TYPE ST_InternalPowerSupply_Params :
STRUCT
	i_ACStartupDelay : INT := 100; //ms
	i_DCPSU_StartupDelay: INT := 1000; //ms
	i_ACPSU_StartupDelay: INT := 1000; //ms
	
	//trigger level before Battery low error is issued. 
	usi_UPSBattLowErrorSOC		:	USINT 	:= 30;
	//UPS charging request was apparently denied. System should shutdown? 
	usi_UPSBattLowwarningSOC	:	USINT 	:= 50;
	//trigger level before Battery low warning is issued and UPS charging is requested from Internal power supply
	LowBatteryShutdownTimer		:	TIME := T#10M;
	
	//Battery self test interval (days). 0 means disable
	t_UPSBattSelfTestInterval	:	TIME := T#30D;
	
END_STRUCT
END_TYPE

(* stored: Version 1.1.0.1, ProductVersion 3.1.4026.18
   DUT ST_InternalPowerSupply_Params: Id {c73dfe6b-5e2f-44ec-bb03-5b9f131c3f99} *)
